FUNCTION_BLOCK FB_AutomaticControl
VAR_INPUT
END_VAR
VAR_OUTPUT
END_VAR
VAR
	fbMotionReferenceGenerator : FB_MotionReferenceGenerator;
END_VAR

fbMotionReferenceGenerator(
	bEnable := TRUE,
	fStartPosition_m := 0.0,
	fStartVelocity_m := 0.0,
	fPositionSetpoint_m := 0.4,
	fVelocitySetpoint_m := 0.05,
	fTimeBeforeStarting_s := 2,
	fRampTime_s := 1,
	fHoldPositionTime_s := 3,
	fClock_s := Parameters.stStateVariables.fTime, 
	fVelocityReference_m => HMI.fCylinderVelocity,
	fPositionReference_m => HMI.fCylinderPositon
);

END_FUNCTION_BLOCK

(* stored: Version 1.1.0.1, ProductVersion 3.1.4024.10
   POU FB_AutomaticControl: Id {64696064-021d-4e51-bf2c-8162c27d0f9f}, SpecialFunc None *)
